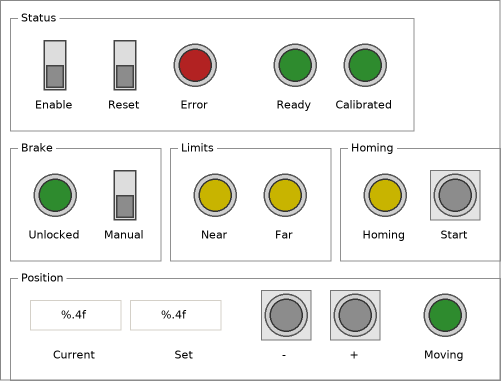
VISUALIZATION Focus  // 501x381
    GroupBox (10,10 404x121), "Status"
        DipSwitch (20,30 50x50), variable: MAIN.FocusControl.bEnable, behaviour: TOGGLE, style: Switch-DipSwitch-Gray
        DipSwitch (90,30 50x50), variable: MAIN.FocusControl.bReset, behaviour: TOGGLE, style: Switch-DipSwitch-Gray
        Lamp1 (160,30 50x50), variable: MAIN.FocusControl.bError, style: Lamp-Lamp1-Red
        Lamp1 (260,30 50x50), variable: MAIN.FocusControl.bReady, style: Lamp-Lamp1-Green
        Lamp1 (330,30 50x50), variable: MAIN.FocusControl.bCalibrated, style: Lamp-Lamp1-Green
        Label (10,80 68x30), "Enable"
        Label (80,80 68x30), "Reset"
        Label (150,80 68x30), "Error"
        Label (250,80 68x30), "Ready"
        Label (320,80 68x30), "Calibrated"
        Lamp1 (410,280 50x50), variable: MAIN.AzimuthControl.bCalibrated, style: Lamp-Lamp1-Green
    GroupBox (340,140 161x121), "Homing"
        Lamp1 (20,30 50x50), variable: MAIN.FocusControl.bHomeAxis, style: Lamp-Lamp1-Yellow
        Label (10,80 68x30), "Homing"
        PushSwitch (90,30 50x50), variable: MAIN.FocusControl.bHomeAxis, behaviour: TOGGLE, style: Switch-PushSwitch-Gray
        Label (80,80 68x30), "Start"
    GroupBox (10,140 151x121), "Brake"
        DipSwitch (90,30 50x50), variable: MAIN.FocusControl.bManualUnlock, behaviour: TOGGLE, style: Switch-DipSwitch-Gray
        Lamp1 (20,30 50x50), variable: MAIN.FocusControl.bFocusUnlocked, style: Lamp-Lamp1-Green
        Label (80,80 68x30), "Manual"
        Label (10,80 68x30), "Unlocked"
    GroupBox (170,140 161x121), "Limits"
        Lamp1 (20,30 50x50), variable: MAIN.FocusControl.IbLimitNear, style: Lamp-Lamp1-Yellow
        Label (10,80 68x30), "Near"
        Lamp1 (90,30 50x50), variable: MAIN.FocusControl.IbLimitFar, style: Lamp-Lamp1-Yellow
    Label (250,220 68x30), "Far"
    GroupBox (10,270 491x111), "Position"
        Textfield (20,30 91x30), "%.4f", text variable: MAIN.FocusControl.fActualPosition
        Label (30,70 68x30), "Current"
        Textfield (120,30 91x30), "%.4f", text variable: MAIN.FocusControl.fPosition
            OnMouseUp: write the text variable via InputWithLimits, min MAIN.AzimuthControl.fMinPosition, max MAIN.AzimuthControl.fMaxPosition
        PushSwitch (251,20 50x50), variable: MAIN.FocusControl.bMoveNeg, behaviour: TOGGLE, style: Switch-PushSwitch-Gray
        PushSwitch (320,20 50x50), variable: MAIN.FocusControl.bMovePos, behaviour: TOGGLE, style: Switch-PushSwitch-Gray
        Label (240,70 68x30), "-"
        Label (310,70 68x30), "+"
        Label (140,70 68x30), "Set"
        Lamp1 (410,20 50x50), variable: MAIN.FocusControl.bMoveAxis, style: Lamp-Lamp1-Green
    Label (410,340 68x30), "Moving"
END_VISUALIZATION

(* stored: Version 1.1.0.1, ProductVersion 3.1.4024.15
   Visu Focus: Id {4c422a0a-5b19-4f69-935a-a6b0140fc755} *)
